{attribute 'GeneratedUsingTerminal: AX8206-0100-0102-0102'}
{attribute addProperty BoxType "AX8206-0100-0102-0102"}
{attribute addProperty Id "DeviceDevice_6E2575772Device_SafetyDevice_Safety_C21945A160Ch_ACh_A_D18C6F1622Ch_BCh_B_647F9A0C22WcStateAT %I*WcState_B516A2644InfoDataAT %I*InfoData_FD1CC0AA12"}
{attribute addProperty CRC "762843330"}
{attribute addProperty Size "122"}
TYPE AX8206_2D7810C2 EXTENDS EtcSlaveTerminalBase_947E5A46 :
STRUCT
	{attribute addProperty Name "Device"}
	Device : Device_6E257577;
	{attribute addProperty Name "Device_Safety"}
	Device_Safety : Device_Safety_C21945A1;
	{attribute addProperty Name "Ch_A"}
	Ch_A : Ch_A_D18C6F16;
	{attribute addProperty Name "Ch_B"}
	Ch_B : Ch_B_647F9A0C;
	{attribute addProperty Name "WcState"}
	WcState : WcState_B516A264;
	{attribute addProperty Name "InfoData"}
	InfoData : InfoData_FD1CC0AA;
END_STRUCT
END_TYPE

(* stored: Version 1.2.0.0, ProductVersion 3.1.4024.9
   DUT AX8206_2D7810C2: Id {a9a5ffdd-70f7-4fd7-aa7f-2449a1e531b4} *)
